// Mitsubishi GX Works2 project: 4   PLC: FX3U/FX3UC

// task Task_01 (event TRUE, interval 0, priority 31): POU_01

PROGRAM POU_01
VAR
  wstep : INT;
  ton1 : TON;
  ii : INT;
END_VAR
IF M8002 THEN
	wstep := 0;
END_IF;

IF M10 THEN
	wstep := 0;
END_IF;

CASE wstep OF 
	0:
	FOR ii := 0 TO 2 BY 1 DO
		Z0 := ii;
		Y0Z0 := FALSE;
	END_FOR;
	ton1(IN := FALSE);

	IF M11 THEN
		wstep := 20;
	END_IF;
	
	20:
	Y2 := FALSE;
	Y0 := TRUE;
	Y1 := TRUE;
	ton1(IN := NOT ton1.Q, PT := T#1s);
	IF ton1.Q THEN
		wstep := 21;		
	END_IF;
	
	21:
	Y0 := FALSE;
	Y2 := TRUE;
	ton1(IN := NOT ton1.Q, PT := T#1s);
	IF ton1.Q THEN
		wstep := 22;
	END_IF;
	
	22:
	Y1 := FALSE;
	Y0 := TRUE;
	ton1(IN := NOT ton1.Q, PT := T#1s);
	IF ton1.Q THEN
		wstep := 20;
	END_IF;	
END_CASE;
END_PROGRAM
